(* CoDeSys 2.3.9.62 project: ascensor_doble_memoria.pro *)
(* Libraries: Standard.lib 2.6.14 10:37:46, IecSfc.lib 2.6.14 11:37:46 *)

(* Global variable list: Global_Variables *)
VAR_GLOBAL
   (*Entradas *)
      (* Sensores de posición en plantas *)
      S0_1: BOOL;
      S1_1: BOOL;
      S2_1: BOOL;
      S3_1: BOOL;
      S0_2: BOOL;
      S1_2: BOOL;
      S2_2: BOOL;
      S3_2: BOOL;
      (* Pulsadores de llamadas en planta *)
      P0: BOOL;
      P1: BOOL;
      P2: BOOL;
      P3: BOOL;
    (* Pulsadores en cabina  *)
      C0_1: BOOL;
      C1_1: BOOL;
      C2_1: BOOL;
      C3_1: BOOL;
      C0_2: BOOL;
      C1_2: BOOL;
      C2_2: BOOL;
      C3_2: BOOL;
   (*Salidas *)
      Motor_arriba_1 : BOOL;
      Motor_Abajo_1 : BOOL;
     Motor_arriba_2 : BOOL;
      Motor_Abajo_2 : BOOL;
   (* luces asociadas a los pulsadores. Se usarán
        si se quiere implementar memoria de llamada *)
     LuzP0:BOOL;
     LuzP1:BOOL;
     LuzP2:BOOL;
     LuzP3:BOOL;
     LuzC0_1:BOOL;
     LuzC1_1:BOOL;
     LuzC2_1:BOOL;
     LuzC3_1:BOOL;
     LuzC0_2:BOOL;
     LuzC1_2:BOOL;
     LuzC2_2:BOOL;
     LuzC3_2:BOOL;
(* otras variables*)
	rearme,emergencia,emer_btn, Luzemer:BOOL;
	TM1:TIME:= T#2s;
	TM2:TIME:=T#3s;

END_VAR

(* POU PLC_PRG, ST *)
PROGRAM PLC_PRG
VAR
	asc1:Ascensor;
END_VAR
Movimiento1;
Movimiento2;
Ascensores_prg;
END_PROGRAM

(* POU Ascensor, SFC *)
FUNCTION_BLOCK Ascensor
VAR_INPUT
	PC0,PC1,PC2,PC3:BOOL;(*Pulsadores internos a la cabina*)
	Selec:BOOL;(*seleccionamos al ascensor para acepte la planta del pulsador externo*)
	EntPulsador:INT;
	PE0,PE1,PE2,PE3:BOOL;(*Pusadores externos ppoporcionados por el controlador*)
	SP0,SP1,SP2,SP3:BOOL;(*Sensores de planta*)
	e,ra:BOOL;(*emergencia y rearme*)
END_VAR
VAR_OUTPUT
	MotorArriba, MotorAbajo:BOOL; (*de aquí deducimos los sentido*)
	(*la puerta la quitamos*)
	LI0:BOOL;
	LI1:BOOL;
	Li2:BOOL;
	Li3:BOOL;
	Adestino: ARRAY [0..4] OF BOOL;(*Arrary de plantas a las que voy a visitar*) (*la idea es que si un ascensor va en ese sentido, el controlador lo añada a la lista de destinos por visitar *)(*la 4 es pplanta no definida*)
	UltimoSentido:BOOL;
END_VAR
VAR
	PA:PlantaActual_FB;
	PlantaActual:INT:=0;
	destEnc:BOOL:=FALSE; (*Indica si ha encontrado un destino*)
	Sentido:BOOL;
	i: INT;
	emer_asc: BOOL;
	luzint: ARRAY [0..3] OF BOOL;

END_VAR
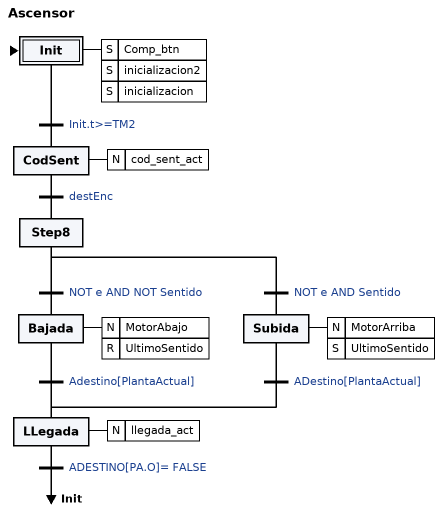
INITIAL_STEP Init:
	Comp_btn(S);
	inicializacion2(S);
	inicializacion(S);
END_STEP
TRANSITION FROM Init TO CodSent := Init.t>=TM2;
END_TRANSITION
STEP CodSent:
	cod_sent_act(N);
END_STEP
TRANSITION FROM CodSent TO Step8 := destEnc;
END_TRANSITION
STEP Step8:
END_STEP
TRANSITION FROM Step8 TO Bajada := NOT e AND NOT Sentido;
END_TRANSITION
TRANSITION FROM Step8 TO Subida := NOT e AND Sentido;
END_TRANSITION
STEP Bajada:
	MotorAbajo(N);
	UltimoSentido(R);
END_STEP
TRANSITION FROM Bajada TO LLegada := Adestino[PlantaActual];
END_TRANSITION
STEP Subida:
	MotorArriba(N);
	UltimoSentido(S);
END_STEP
TRANSITION FROM Subida TO LLegada := ADestino[PlantaActual];
END_TRANSITION
STEP LLegada:
	llegada_act(N);
END_STEP
TRANSITION FROM LLegada TO Init := ADESTINO[PA.O]= FALSE;
END_TRANSITION
END_FUNCTION_BLOCK
ACTION cod_sent_act:
(* deberia ser una funcion*)
    IF sentido AND NOT (Sp3) THEN (* Subida *)
        FOR i := PA.o + 1 TO 3 DO
            IF Adestino[i] THEN
                destEnc:=TRUE;


                EXIT;
            END_IF;
        END_FOR;
    ELSIF NOT SP0 AND NOT Sentido THEN
        FOR i := PA.o - 1 TO 0 BY -1 DO
            IF Adestino[i] THEN
                destEnc:=TRUE;


                EXIT;
            END_IF;
        END_FOR;
    END_IF;

    (* Si no encontró, cambiar el sentido y repetir la búsqueda *)
    IF  NOT destEnc THEN
        sentido := NOT sentido;

        IF sentido AND NOT (Sp3)  THEN (* Subida *)
            FOR i := PA.o + 1 TO 3 DO
                IF Adestino[i] THEN
                    destEnc := TRUE;

                    EXIT;
                END_IF;
            END_FOR;
        ELSIF NOT (Sp0) AND NOT Sentido THEN
            FOR i := PA.o - 1 TO 0 BY -1 DO
                IF Adestino[i] THEN
                    destEnc := TRUE;
                    EXIT;
                END_IF;
            END_FOR;
        END_IF;
    END_IF;
END_ACTION
ACTION Comp_btn:
(*se encarga de añadir los nuevos destinos, otros casos los ignora*)
(* no se puede añadir una planta a la memoria si ya estoy parado  en ella o hay una emergencia *)
(*si estoy parado en esa planta -> otro caso (se vuelven a abrir las puertas)*)
(* sse pulsa ubn boton de la propia cabina cuando se o un boton externo*)

IF NOT e THEN
(* multiples ifs independiente por si se pulsan varios botones a la vez*)
(* aunque debido a los limites de la simulacion esto no pasa *)
	IF  NOT (SP0 AND NOT MotorArriba AND NOT MotorAbajo) AND (PC0 OR PE0) THEN
	Adestino[0]:=TRUE;
	luzint[0]:= PC0 OR luzint[0];
	END_IF
	IF  NOT (SP1 AND NOT MotorArriba AND NOT MotorAbajo) AND (PC1 OR PE1) THEN
	Adestino[1]:=TRUE;
	luzint[1]:= PC1 OR luzint[1];
	END_IF
	IF  NOT (SP2 AND NOT MotorArriba AND NOT MotorAbajo) AND (PC2 OR PE2) THEN
	Adestino[2]:=TRUE;
	luzint[2]:= PC2 OR luzint[2];
	END_IF
	IF  NOT (SP3 AND NOT MotorArriba AND NOT MotorAbajo) AND (PC3 OR PE3) THEN
	Adestino[3]:=TRUE;
	luzint[3]:= PC3 OR luzint[3];
	END_IF
END_IF
END_ACTION
ACTION inicializacion:
Pa(S0:=SP0,S1:=SP1,S2:=SP2,S3:=SP3, O=>PlantaActual);
END_ACTION
ACTION inicializacion2:
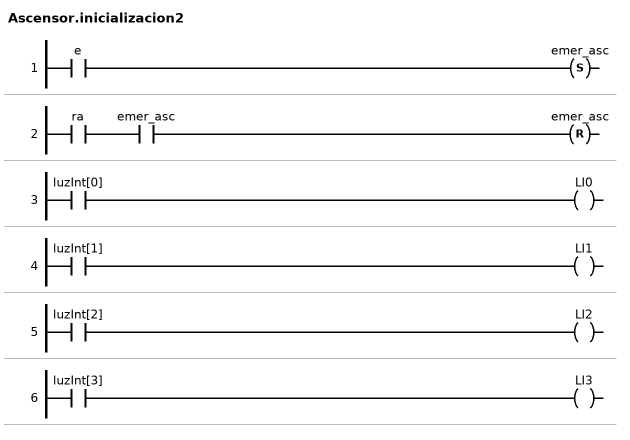
_LD_ (* Ladder Diagram *)
NETWORK 1
	[e] --- (S emer_asc)
NETWORK 2
	[ra] - [emer_asc] --- (R emer_asc)
NETWORK 3
	[luzInt[0]] --- (LI0)
NETWORK 4
	[luzInt[1]] --- (LI1)
NETWORK 5
	[luzInt[2]] --- (LI2)
NETWORK 6
	[luzInt[3]] --- (LI3)
_END_LD_
(* the same logic as Structured Text *)
(* Network 1 *)
IF e THEN emer_asc := TRUE; END_IF;
(* Network 2 *)
IF ra AND emer_asc THEN emer_asc := FALSE; END_IF;
(* Network 3 *)
LI0 := luzInt[0];
(* Network 4 *)
LI1 := luzInt[1];
(* Network 5 *)
LI2 := luzInt[2];
(* Network 6 *)
LI3 := luzInt[3];
END_ACTION
ACTION llegada_act:
destEnc:=FALSE;
luzInt[PlantaActual]:=FALSE;
Adestino[PlantaActual]:=FALSE;
END_ACTION

(* POU PlantaActual_FB, ST *)
FUNCTION_BLOCK PlantaActual_FB
VAR_INPUT
	S0,S1,S2,S3:BOOL;
END_VAR
VAR_OUTPUT
	O:INT;
END_VAR
VAR
END_VAR
IF(S0) THEN
O:=0;
ELSIF S1 THEN
o:= 1;
ELSIF S2 THEN
o:=2;
ELSIF S3 THEN
o:= 3;
ELSE  o:=4;
(*La planta no existente*)
END_IF
END_FUNCTION_BLOCK

(* POU Movimiento1, ST *)
PROGRAM Movimiento1
VAR
    pos1:INT:=0;
END_VAR
IF (Motor_arriba_1 AND pos1>=-240) THEN
   pos1:=pos1-2;
END_IF


IF (Motor_abajo_1 AND pos1<=-2) THEN
   pos1:=pos1+2;
END_IF

IF (pos1>=0 AND pos1<=2) THEN
  S0_1:=TRUE;
ELSE
  S0_1:=FALSE;
END_IF

IF (pos1>=-78 AND pos1<=-74) THEN
  S1_1:=TRUE;
ELSE
  S1_1:=FALSE;
END_IF

IF (pos1>=-156 AND pos1<=-152) THEN
  S2_1:=TRUE;
ELSE
  S2_1:=FALSE;
END_IF

IF (pos1>=-242 AND pos1<=-240) THEN
  S3_1:=TRUE;
ELSE
  S3_1:=FALSE;
END_IF
END_PROGRAM

(* POU Movimiento2, ST *)
PROGRAM Movimiento2
VAR
    pos2:INT:=0;
END_VAR
IF (Motor_arriba_2 AND pos2>=-240) THEN
   pos2:=pos2-2;
END_IF


IF (Motor_abajo_2 AND pos2<=-2) THEN
   pos2:=pos2+2;
END_IF

IF (pos2>=0 AND pos2<=2) THEN
  S0_2:=TRUE;
ELSE
  S0_2:=FALSE;
END_IF

IF (pos2>=-78 AND pos2<=-74) THEN
  S1_2:=TRUE;
ELSE
  S1_2:=FALSE;
END_IF

IF (pos2>=-156 AND pos2<=-152) THEN
  S2_2:=TRUE;
ELSE
  S2_2:=FALSE;
END_IF

IF (pos2>=-242 AND pos2<=-240) THEN
  S3_2:=TRUE;
ELSE
  S3_2:=FALSE;
END_IF
END_PROGRAM

(* POU Ascensores_prg, LD *)
PROGRAM Ascensores_prg
VAR
	Asc1: Ascensor;
	Asc2: Ascensor;
	cntrllr: controller;
END_VAR
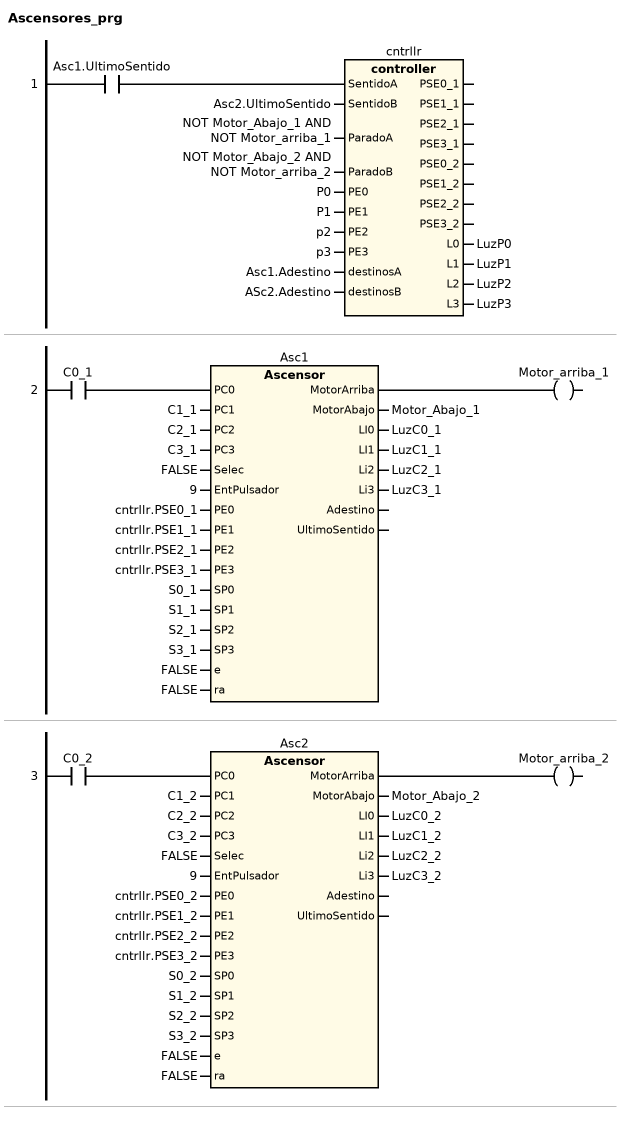
_LD_ (* Ladder Diagram *)
NETWORK 1
	[Asc1.UltimoSentido] - cntrllr:controller(SentidoA: *, SentidoB: Asc2.UltimoSentido, ParadoA: NOT Motor_Abajo_1 AND NOT Motor_arriba_1, ParadoB: NOT Motor_Abajo_2 AND NOT Motor_arriba_2, PE0: P0, PE1: P1, PE2: p2, PE3: p3, destinosA: Asc1.Adestino, destinosB: ASc2.Adestino, L0 => LuzP0, L1 => LuzP1, L2 => LuzP2, L3 => LuzP3)
NETWORK 2
	[C0_1] - Asc1:Ascensor(PC0: *, PC1: C1_1, PC2: C2_1, PC3: C3_1, Selec: FALSE, EntPulsador: 9, PE0: cntrllr.PSE0_1, PE1: cntrllr.PSE1_1, PE2: cntrllr.PSE2_1, PE3: cntrllr.PSE3_1, SP0: S0_1, SP1: S1_1, SP2: S2_1, SP3: S3_1, e: FALSE, ra: FALSE, MotorAbajo => Motor_Abajo_1, LI0 => LuzC0_1, LI1 => LuzC1_1, Li2 => LuzC2_1, Li3 => LuzC3_1) --- (Motor_arriba_1)
NETWORK 3
	[C0_2] - Asc2:Ascensor(PC0: *, PC1: C1_2, PC2: C2_2, PC3: C3_2, Selec: FALSE, EntPulsador: 9, PE0: cntrllr.PSE0_2, PE1: cntrllr.PSE1_2, PE2: cntrllr.PSE2_2, PE3: cntrllr.PSE3_2, SP0: S0_2, SP1: S1_2, SP2: S2_2, SP3: S3_2, e: FALSE, ra: FALSE, MotorAbajo => Motor_Abajo_2, LI0 => LuzC0_2, LI1 => LuzC1_2, Li2 => LuzC2_2, Li3 => LuzC3_2) --- (Motor_arriba_2)
_END_LD_
(* the same logic as Structured Text *)
(* Network 1 *)
cntrllr(SentidoA := Asc1.UltimoSentido, SentidoB := Asc2.UltimoSentido, ParadoA := NOT Motor_Abajo_1 AND NOT Motor_arriba_1, ParadoB := NOT Motor_Abajo_2 AND NOT Motor_arriba_2, PE0 := P0, PE1 := P1, PE2 := p2, PE3 := p3, destinosA := Asc1.Adestino, destinosB := ASc2.Adestino);
LuzP0 := cntrllr.L0;
LuzP1 := cntrllr.L1;
LuzP2 := cntrllr.L2;
LuzP3 := cntrllr.L3;
(* Network 2 *)
Asc1(PC0 := C0_1, PC1 := C1_1, PC2 := C2_1, PC3 := C3_1, Selec := FALSE, EntPulsador := 9, PE0 := cntrllr.PSE0_1, PE1 := cntrllr.PSE1_1, PE2 := cntrllr.PSE2_1, PE3 := cntrllr.PSE3_1, SP0 := S0_1, SP1 := S1_1, SP2 := S2_1, SP3 := S3_1, e := FALSE, ra := FALSE);
Motor_Abajo_1 := Asc1.MotorAbajo;
LuzC0_1 := Asc1.LI0;
LuzC1_1 := Asc1.LI1;
LuzC2_1 := Asc1.Li2;
LuzC3_1 := Asc1.Li3;
Motor_arriba_1 := Asc1.MotorArriba;
(* Network 3 *)
Asc2(PC0 := C0_2, PC1 := C1_2, PC2 := C2_2, PC3 := C3_2, Selec := FALSE, EntPulsador := 9, PE0 := cntrllr.PSE0_2, PE1 := cntrllr.PSE1_2, PE2 := cntrllr.PSE2_2, PE3 := cntrllr.PSE3_2, SP0 := S0_2, SP1 := S1_2, SP2 := S2_2, SP3 := S3_2, e := FALSE, ra := FALSE);
Motor_Abajo_2 := Asc2.MotorAbajo;
LuzC0_2 := Asc2.LI0;
LuzC1_2 := Asc2.LI1;
LuzC2_2 := Asc2.Li2;
LuzC3_2 := Asc2.Li3;
Motor_arriba_2 := Asc2.MotorArriba;
END_PROGRAM

(* POU controller, SFC *)
FUNCTION_BLOCK controller
VAR_INPUT
	SentidoA,SentidoB:BOOL;
	ParadoA,ParadoB:BOOL;
	PE0,PE1,PE2,PE3:BOOL;(*Entradas del pulsador externo*)
	destinosA, destinosB: ARRAY [0..4] OF BOOL;(*Arrays de destino de los ascensors*)
END_VAR
VAR_OUTPUT
	PSE0_1,PSE1_1,PSE2_1,PSE3_1:BOOL;
	PSE0_2,PSE1_2,PSE2_2,PSE3_2:BOOL;
	L0,L1,L2,L3:BOOL;
END_VAR
VAR
	btn_pulsado:BOOL:=FALSE;
	valor_btn:INT;
	PE:PulsadorEncoder;
	SelecA: BOOL;
	Lista:BOOL:=FALSE;
	PDA: PulsadorDecoder;
	PDB: PulsadorDecoder;
  	aluces:ARRAY [0..4] OF BOOL;
	Pa: PlantaActual_FB;
	Pb: PlantaActual_FB;
	PlantaA,PlantaB:INT;
	Env_A,ENv_B:BOOL;
END_VAR
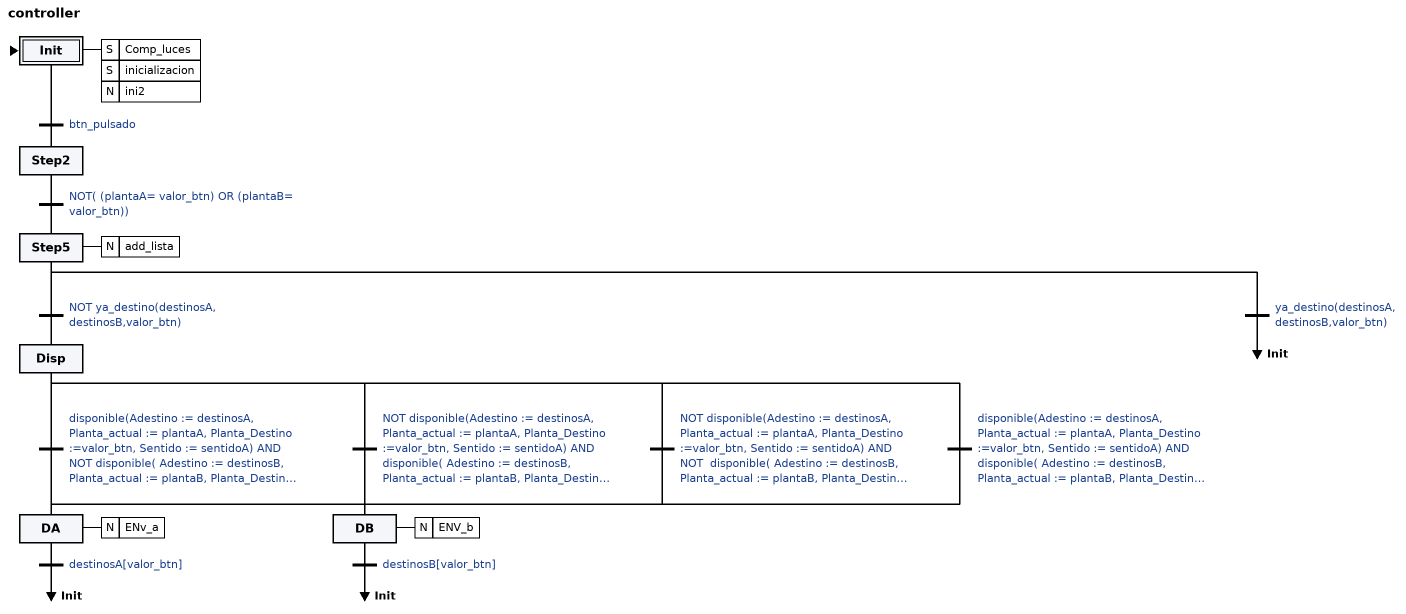
INITIAL_STEP Init:
	Comp_luces(S);
	inicializacion(S);
	ini2(N);
END_STEP
TRANSITION FROM Init TO Step2 := btn_pulsado;
END_TRANSITION
STEP Step2:
END_STEP
TRANSITION FROM Step2 TO Step5 := NOT( (plantaA= valor_btn) OR (plantaB= valor_btn));
END_TRANSITION
STEP Step5:
	add_lista(N);
END_STEP
TRANSITION FROM Step5 TO Disp := NOT ya_destino(destinosA, destinosB,valor_btn);
END_TRANSITION
TRANSITION FROM Step5 TO Init := ya_destino(destinosA, destinosB,valor_btn);
END_TRANSITION
STEP Disp:
END_STEP
TRANSITION FROM Disp TO DA := disponible(Adestino := destinosA, Planta_actual := plantaA, Planta_Destino :=valor_btn, Sentido := sentidoA) AND NOT disponible( Adestino := destinosB, Planta_actual := plantaB, Planta_Destino := valor_btn, Sentido := sentidob);
END_TRANSITION
TRANSITION FROM Disp TO DB := NOT disponible(Adestino := destinosA, Planta_actual := plantaA, Planta_Destino :=valor_btn, Sentido := sentidoA) AND  disponible( Adestino := destinosB, Planta_actual := plantaB, Planta_Destino := valor_btn, Sentido := sentidob);
END_TRANSITION
TRANSITION FROM Disp TO DB := NOT disponible(Adestino := destinosA, Planta_actual := plantaA, Planta_Destino :=valor_btn, Sentido := sentidoA) AND  NOT  disponible( Adestino := destinosB, Planta_actual := plantaB, Planta_Destino := valor_btn, Sentido := sentidob);
END_TRANSITION
TRANSITION FROM Disp TO DA := disponible(Adestino := destinosA, Planta_actual := plantaA, Planta_Destino :=valor_btn, Sentido := sentidoA) AND disponible( Adestino := destinosB, Planta_actual := plantaB, Planta_Destino := valor_btn, Sentido := sentidob);
END_TRANSITION
STEP DA:
	ENv_a(N);
END_STEP
TRANSITION FROM DA TO Init := destinosA[valor_btn];
END_TRANSITION
STEP DB:
	ENV_b(N);
END_STEP
TRANSITION FROM DB TO Init := destinosB[valor_btn];
END_TRANSITION
END_FUNCTION_BLOCK
ACTION add_lista:
aluces[valor_btn]:=TRUE;
END_ACTION
ACTION comp_luces:
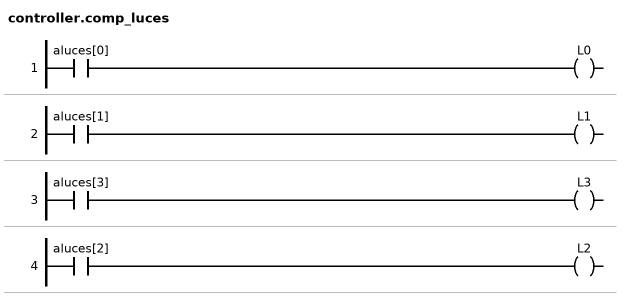
_LD_ (* Ladder Diagram *)
NETWORK 1
	[aluces[0]] --- (L0)
NETWORK 2
	[aluces[1]] --- (L1)
NETWORK 3
	[aluces[3]] --- (L3)
NETWORK 4
	[aluces[2]] --- (L2)
_END_LD_
(* the same logic as Structured Text *)
(* Network 1 *)
L0 := aluces[0];
(* Network 2 *)
L1 := aluces[1];
(* Network 3 *)
L3 := aluces[3];
(* Network 4 *)
L2 := aluces[2];
END_ACTION
ACTION ini2:
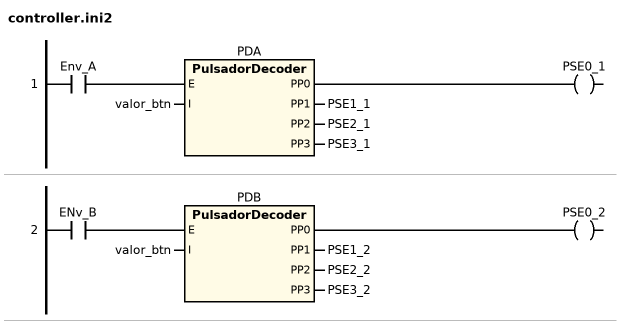
_LD_ (* Ladder Diagram *)
NETWORK 1
	[Env_A] - PDA:PulsadorDecoder(E: *, I: valor_btn, PP1 => PSE1_1, PP2 => PSE2_1, PP3 => PSE3_1) --- (PSE0_1)
NETWORK 2
	[ENv_B] - PDB:PulsadorDecoder(E: *, I: valor_btn, PP1 => PSE1_2, PP2 => PSE2_2, PP3 => PSE3_2) --- (PSE0_2)
_END_LD_
(* the same logic as Structured Text *)
(* Network 1 *)
PDA(E := Env_A, I := valor_btn);
PSE1_1 := PDA.PP1;
PSE2_1 := PDA.PP2;
PSE3_1 := PDA.PP3;
PSE0_1 := PDA.PP0;
(* Network 2 *)
PDB(E := ENv_B, I := valor_btn);
PSE1_2 := PDB.PP1;
PSE2_2 := PDB.PP2;
PSE3_2 := PDB.PP3;
PSE0_2 := PDB.PP0;
END_ACTION
ACTION inicializacion:
PE(PP0:=P0,PP1:=P1,PP2:=P2,PP3:=P3, E=>btn_pulsado);
Pa(S0:=S0_1,S1:=S1_1,S2:=S2_1,S3:=S3_1, O=>PlantaA);
Pb(S0:=S0_2,S1:=S1_2,S2:=S2_2,S3:=S3_2, O=>PlantaB);
IF(btn_pulsado) THEN
valor_btn:= PE.N;
END_IF
IF(ParadoA ) THEN
aluces[PlantaA]:=FALSE;
END_IF
IF(ParadoB) THEN
aluces[PlantaB]:=FALSE;
END_IF
END_ACTION

(* POU PulsadorEncoder, ST *)
FUNCTION_BLOCK PulsadorEncoder
VAR_INPUT
	PP0,PP1,PP2,PP3:BOOL;
END_VAR
VAR_OUTPUT
	N:INT; (*Si vale 4 no vale*)
	E:BOOL;
END_VAR
VAR
END_VAR
E:= PP0 OR PP1 OR PP2 OR PP3;
IF E THEN
IF PP0 THEN
N:=0;
ELSIF PP1 THEN
N:=1;
ELSIF PP2 THEN
N:=2;
ELSIF PP3 THEN
N:=3;
END_IF
END_IF
END_FUNCTION_BLOCK

(* POU PulsadorDecoder, ST *)
FUNCTION_BLOCK PulsadorDecoder
VAR_INPUT
	E: BOOL;
	I:INT;
END_VAR
VAR_OUTPUT
	PP0,PP1,PP2,PP3:BOOL;
END_VAR
VAR
	RT: R_TRIG;
END_VAR
IF E THEN
CASE I OF
0: PP0:=TRUE;
1: PP1:= TRUE;
2: PP2:=TRUE;
3: PP3:=TRUE;
END_CASE
ELSE
PP0:=FALSE;
PP1:=FALSE;
PP3:=FALSE;
PP0:=FALSE;
END_IF
END_FUNCTION_BLOCK

(* POU ya_destino, ST *)
FUNCTION ya_destino : BOOL
VAR_INPUT
	destinosA, destinosb: ARRAY [0..4] OF BOOL;(*Arrays de destino de los ascensors*)
	planta_solicitada:INT;
END_VAR
VAR
END_VAR
(*devuelve true si el destino esta asignado a una de las listas*)
IF destinosA[planta_solicitada] OR destinosB[planta_solicitada] AND planta_solicitada <=3 AND Planta_solicitada>=0 THEN
    ya_destino := TRUE;
ELSE ya_destino:=FALSE;
END_IF
END_FUNCTION

(* POU disponible, ST *)
FUNCTION disponible : BOOL
VAR_INPUT
	 Adestino: ARRAY [0..4] OF BOOL;
	Planta_actual:INT;
	Planta_Destino:INT;
	Sentido:BOOL;
END_VAR
VAR
    i : INT;
    tiene_destinos : BOOL;
    sentido_favorable : BOOL;
END_VAR
(* 1. Verificar si el ascensor tiene destinos activos *)
tiene_destinos := FALSE;
FOR i := 0 TO 4 DO
    IF Adestino[i] THEN
        tiene_destinos := TRUE;
        EXIT;
    END_IF;
END_FOR;

(* 2. Verificar si el sentido es favorable a la planta destino *)
IF Sentido = TRUE THEN
    sentido_favorable := Planta_Destino > Planta_actual;
ELSE
    sentido_favorable := Planta_Destino < Planta_actual;
END_IF;

(* 3. Devolver disponibilidad *)
IF NOT tiene_destinos THEN
    disponible := TRUE;
ELSIF sentido_favorable THEN
    disponible := TRUE;
ELSE
    disponible := FALSE;
END_IF;
END_FUNCTION

(* Visualisation Ascensor
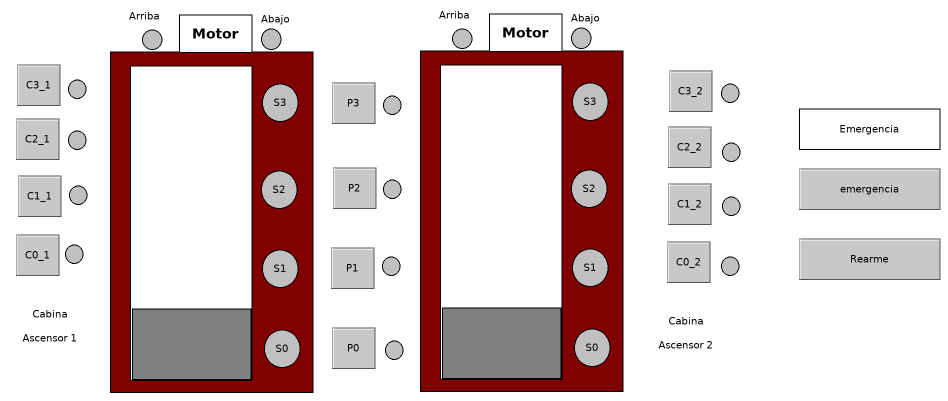
ellipse at (285,341)-(321,379): text "S0"; alarm colour if S0_1
ellipse at (283,261)-(319,299): text "S1"; alarm colour if S1_1
ellipse at (282,182)-(318,220): text "S2"; alarm colour if S2_1
ellipse at (283,95)-(319,133): text "S3"; alarm colour if S3_1
rounded rectangle at (153,320)-(272,391): y offset Movimiento1.pos1
button at (353,339)-(396,380): text "P0"; taps P0
button at (352,259)-(395,300): text "P1"; taps P1
button at (354,179)-(397,220): text "P2"; taps P2
button at (353,94)-(396,135): text "P3"; taps P3
rectangle at (200,26)-(273,64): text "Motor"
ellipse at (163,41)-(183,61): alarm colour if Motor_arriba_1
ellipse at (282,40)-(302,61): alarm colour if Motor_abajo_1
rectangle at (138,18)-(193,37): text "Arriba"
rectangle at (269,21)-(324,40): text "Abajo"
ellipse at (595,340)-(631,378): text "S0"; alarm colour if S0_2
ellipse at (593,260)-(629,298): text "S1"; alarm colour if S1_2
ellipse at (592,181)-(628,219): text "S2"; alarm colour if S2_2
ellipse at (593,94)-(629,132): text "S3"; alarm colour if S3_2
rounded rectangle at (463,319)-(582,390): y offset Movimiento2.pos2
rectangle at (510,25)-(583,63): text "Motor"
ellipse at (473,40)-(493,60): alarm colour if Motor_arriba_2
ellipse at (592,39)-(612,60): alarm colour if Motor_abajo_2
rectangle at (448,17)-(503,36): text "Arriba"
rectangle at (579,20)-(634,39): text "Abajo"
button at (37,246)-(80,287): text "C0_1"; taps C0_1
button at (39,187)-(82,228): text "C1_1"; taps C1_1
button at (37,130)-(80,171): text "C2_1"; taps C2_1
button at (38,76)-(81,117): text "C3_1"; taps C3_1
rectangle at (28,305)-(114,346): text "Cabina"
rectangle at (28,329)-(114,370): text "Ascensor 1"
button at (688,253)-(731,294): text "C0_2"; taps C0_2
button at (689,195)-(732,236): text "C1_2"; taps C1_2
button at (689,138)-(732,179): text "C2_2"; taps C2_2
button at (690,82)-(733,123): text "C3_2"; taps C3_2
rectangle at (664,312)-(750,353): text "Cabina"
rectangle at (664,336)-(750,377): text "Ascensor 2"
ellipse at (89,91)-(107,110): alarm colour if LuzC3_1
ellipse at (89,142)-(107,161): alarm colour if LuzC2_1
ellipse at (90,197)-(108,216): alarm colour if LuzC1_1
ellipse at (86,256)-(104,275): alarm colour if LuzC0_1
ellipse at (404,107)-(422,126): alarm colour if LuzP3
ellipse at (404,191)-(422,210): alarm colour if LuzP2
ellipse at (403,268)-(421,287): alarm colour if LuzP1
ellipse at (406,352)-(424,371): alarm colour if LuzP0
ellipse at (742,95)-(760,114): alarm colour if LuzC3_2
ellipse at (743,154)-(761,173): alarm colour if LuzC2_2
ellipse at (743,208)-(761,227): alarm colour if LuzC1_2
ellipse at (742,268)-(760,287): alarm colour if LuzC0_2
rectangle at (820,120)-(961,161): text "Emergencia"; taps luzemer
button at (820,180)-(961,221): text "emergencia"; taps emer_btn
button at (820,250)-(961,291): text "Rearme"; taps rearme
6 more shapes without text or variables
*)
